// TIA Portal V17 export
// export: Created 2023-02-26T22:28:46.5168673Z, ExportSetting WithDefaults, DisplayName Totally Integrated Automation Portal, DisplayVersion V17, DisplayName TIA Portal Openness, DisplayVersion V17, DisplayName TIA Portal Version Control Interface, DisplayVersion V17, DisplayName TIA Portal Test Suite Advanced, DisplayVersion V17, DisplayName STEP 7 Professional, DisplayVersion V17, DisplayName SIMATIC Energy Suite, DisplayVersion V17, DisplayName STEP 7 Safety, DisplayVersion V17, DisplayName WinCC Professional, DisplayVersion V17
DATA_BLOCK "ERR_ErrorData"   // DB27
{ S7_Optimized_Access := 'TRUE' }
VERSION : 0.1
// stored: AutoNumber true, IsOnlyStoredInLoadMemory false, IsRetainMemResEnabled false, IsWriteProtectedInAS false, MemoryReserve 100
   VAR
      ErrorChangeMode : Bool;
      ErrorEmergencyStop : Bool;
      ErrorLostPackage_B { S7_SetPoint := 'True'} : Bool;
      ErrorLostPackage : "stt_LostPackageError";
   END_VAR
BEGIN
END_DATA_BLOCK
